Staubli VAL3: extractRow.pgx

public program extractRow(num& x_nInput[] (dimensions=2), num x_nRow, num& x_nResult[])
  local num l_nCol
  local num l_nCounter
  local num l_nRow
begin

  resize(x_nResult,1,1)
  x_nResult = 0
  resize(x_nResult,1, size(x_nInput,2))

  l_nCounter=0
  for l_nCol = 0 to size(x_nInput,2)-1
    x_nResult[l_nCounter] = x_nInput[x_nRow,l_nCol]
    l_nCounter = l_nCounter +1
  endFor

end
